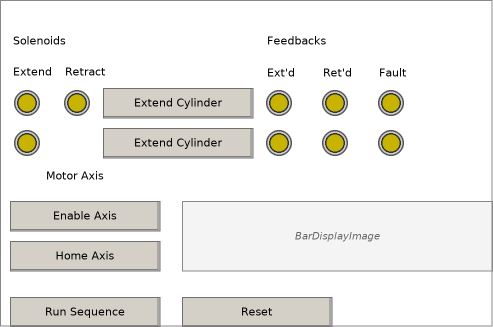
VISUALIZATION Visualization  // 493x327
    Button (103,88 150x30), "Extend Cylinder"
        toggle MAIN.fbVisu.bButtonExtendDouble
    Lamp1 (62,88 30x30), variable: MAIN.fbMachine.fbEquipmentModule1.CylinderDoubleActing._cmdRetract, style: Lamp-Lamp1-Yellow
    Lamp1 (12,88 30x30), variable: MAIN.fbMachine.fbEquipmentModule1.CylinderDoubleActing._cmdExtend, style: Lamp-Lamp1-Yellow
    Lamp1 (320,88 30x30), variable: (MAIN.fbMachine.fbEquipmentModule1.CylinderDoubleActing._state=E_CylinderState.RETRACTED), style: Lamp-Lamp1-Yellow
    Lamp1 (264,88 30x30), variable: (MAIN.fbMachine.fbEquipmentModule1.CylinderDoubleActing._state=E_CylinderState.EXTENDED), style: Lamp-Lamp1-Yellow
    Button (103,128 150x30), "Extend Cylinder"
        toggle MAIN.fbVisu.bButtonExtendSingle
    Lamp1 (12,128 30x30), variable: MAIN.fbMachine.fbEquipmentModule1.CylinderSingleActing._cmdExtend, style: Lamp-Lamp1-Yellow
    Lamp1 (320,128 30x30), variable: (MAIN.fbMachine.fbEquipmentModule1.CylinderSingleActing._state=E_CylinderState.RETRACTED), style: Lamp-Lamp1-Yellow
    Lamp1 (264,128 30x30), variable: (MAIN.fbMachine.fbEquipmentModule1.CylinderSingleActing._state=E_CylinderState.EXTENDED), style: Lamp-Lamp1-Yellow
    Button (10,297 150x30), "Run Sequence"
        toggle MAIN.fbVisu.bButtonRunProduction
    Button (182,297 150x30), "Reset"
        toggle MAIN.fbVisu.bButtonReset
    BarDisplayImage (182,201 311x70), value: MAIN.fbMachine.fbEquipmentModule1.fbAxis1._axis.NcToPlc.ActPos, style: BarDisplayImage-Gray, scale format: %.1f, scale 0..100
    Button (10,201 150x30), "Enable Axis"
        toggle MAIN.fbVisu.bButtonEnableAxis
    Button (10,241 150x30), "Home Axis"
        toggle MAIN.fbVisu.bButtonHomeAxis
    Label (264,26 70x30), "Feedbacks"
    Label (10,26 70x30), "Solenoids"
    Label (0,161 150x30), "Motor Axis"
    Label (10,57 45x30), "Extend"
    Label (62,57 55x30), "Retract"
    Label (320,58 62x30), "Ret'd"
    Label (264,58 64x30), "Ext'd"
    Lamp1 (376,88 30x30), variable: MAIN.fbMachine.fbEquipmentModule1.CylinderDoubleActing._isFaulted, style: Lamp-Lamp1-Yellow
    Label (376,58 62x30), "Fault"
    Lamp1 (376,128 30x30), variable: MAIN.fbMachine.fbEquipmentModule1.CylinderSingleActing._isFaulted, style: Lamp-Lamp1-Yellow
END_VISUALIZATION

(* stored: Version 1.1.0.1, ProductVersion 3.1.4026.18
   Visu Visualization: Id {2f7ac427-d9a4-4b39-a880-4ab6f0692f4b} *)
